// Mitsubishi GX Works2 project: exercicio T0 pulse   PLC: Q03UDV

PROGRAM MAIN
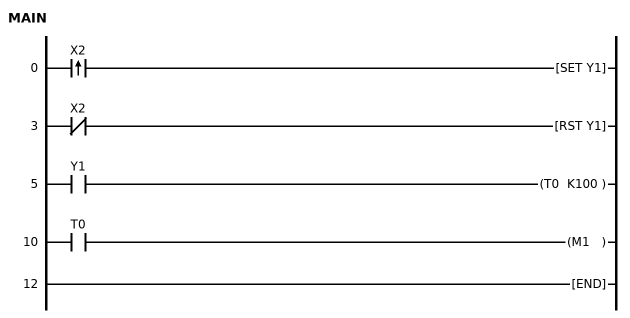
0     LDP     X2
      SET     Y1
3     LDI     X2
      RST     Y1
5     LD      Y1
      OUT     T0 K100
10    LD      T0
      OUT     M1
12    END
END_PROGRAM
